(* IEC 61131-3 sources: test/Class/_OsziLSEBackground, 1 file *)

(* ---- _OsziLSEBackground.st ---- *)
(*!
<Class
	Name               = "_OsziLSEBackground"
	Revision           = "0.0"
	RealtimeTask       = "false"
	CyclicTask         = "false"
	BackgroundTask     = "true"
	Sigmatek           = "true"
	OSInterface        = "false"
	HighPriority       = "false"
	Automatic          = "false"
	UpdateMode         = "Prescan"
	SharedCommandTable = "true"
	Objectsize         = "(284,120)">
	<Channels>
		<Server Name="Server0" Visualized="true" Initialize="false" WriteProtected="true" Retentive="false"/>
	</Channels>
</Class>
*)
_OsziLSEBackground : CLASS
  //Servers:
	Server0 	: SvrChCmd_DINT;
  //Clients:
  //Variables:
		LseOszi 	: ^_LSEOSZI;
  //Functions:

	FUNCTION _OsziLSEBackground
		VAR_OUTPUT
			ret_code 	: ConfStates;
		END_VAR;

	FUNCTION VIRTUAL GLOBAL Background
		VAR_INPUT
			EAX 	: UDINT;
		END_VAR
		VAR_OUTPUT
			state (EAX) 	: UDINT;
		END_VAR;

	FUNCTION GLOBAL PutPtr
		VAR_INPUT
			pLseOszi 	: ^_LSEOSZI;
		END_VAR;
  //Tables:
	FUNCTION @STD
		VAR_OUTPUT
			ret_code	: CONFSTATES;
		END_VAR;
	FUNCTION GLOBAL TAB @CT_;
END_CLASS;

//*********************Inserted from .\_OsziLSEBackground\_OsziLSEBackground_00_00.st*********************

FUNCTION  _OsziLSEBackground::_OsziLSEBackground
VAR_OUTPUT
	ret_code		: CONFSTATES;
END_VAR

  LseOszi := NIL;

	ret_code	:= C_OK;

END_FUNCTION //  _OsziLSEBackground::_OsziLSEBackground

FUNCTION VIRTUAL GLOBAL _OsziLSEBackground::Background
VAR_INPUT
	EAX		: UDINT;
END_VAR
VAR_OUTPUT
	state		: UDINT;
END_VAR

  if(LseOszi <> NIL) then
    LseOsziCyclic(LseOszi);
  end_if;

  state := READY$UDINT;

END_FUNCTION //VIRTUAL GLOBAL _OsziLSEBackground::Background

FUNCTION GLOBAL _OsziLSEBackground::PutPtr
VAR_INPUT
	pLseOszi		: ^_LSEOSZI;
END_VAR

  LseOszi := pLseOszi;

END_FUNCTION //GLOBAL _OsziLSEBackground::PutPtr
